(* PLC project CALENDARS, Actility iec61131 1.0.24, author Laurent Nicq *)
(* stored: creationDateTime 2013-03-20T17:09:43, version 1.0.1, modificationDateTime 2013-07-25T17:16:31 *)

PROGRAM Calendar_Single
  VAR
    Light_Outside : BOOL;
  END_VAR
  VAR_EXTERNAL
    TimeSTART_Single : TOD;
    TimeEND_Single : TOD;
    Date_Single : DATE;
  END_VAR
  VAR
    Calendar_Name : STRING := 'Evening';
  END_VAR

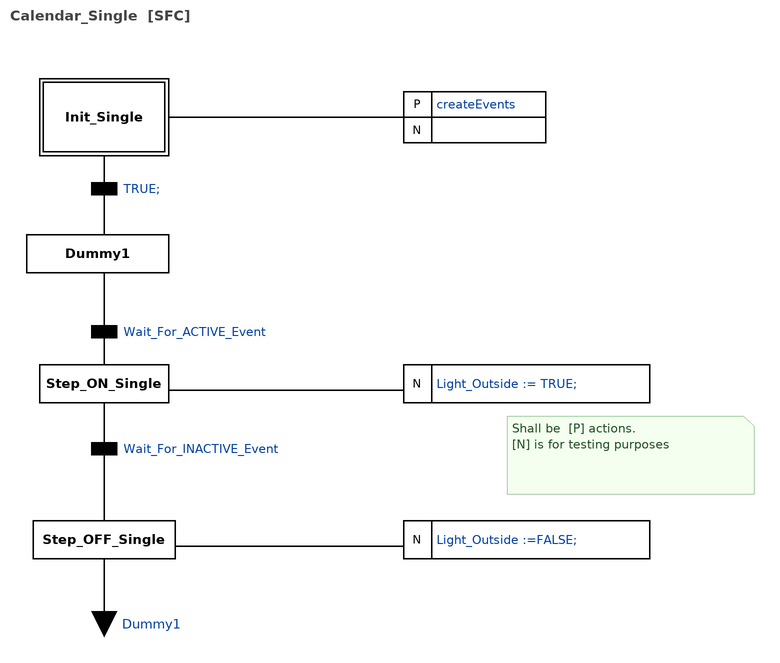
(* Shall be  [P] actions.
[N] is for testing purposes *)
INITIAL_STEP Init_Single:
  createEvents(P);
  (N);
END_STEP
TRANSITION FROM Init_Single TO Dummy1
  := TRUE;
END_TRANSITION
STEP Dummy1:
END_STEP
TRANSITION FROM Dummy1 TO Step_ON_Single  (* Wait_For_ACTIVE_Event *)
  := checkCalendarEvent (Calendar_Name);
END_TRANSITION
STEP Step_ON_Single:
  STEP_ON_SINGLE_INLINE1(N);
END_STEP
ACTION STEP_ON_SINGLE_INLINE1:
  Light_Outside := TRUE;
END_ACTION
TRANSITION FROM Step_ON_Single TO Step_OFF_Single  (* Wait_For_INACTIVE_Event *)
  := NOT(checkCalendarEvent (Calendar_Name) );
END_TRANSITION
STEP Step_OFF_Single:
  STEP_OFF_SINGLE_INLINE2(N);
END_STEP
ACTION STEP_OFF_SINGLE_INLINE2:
  Light_Outside :=FALSE;
END_ACTION

ACTION createEvents:
TimeEND_Single := ADD_TOD_TIME( TimeSTART_Single, T#1m0s);
newCalendarEvent (Calendar_Name, Date_Single, TimeSTART_Single, TimeEND_Single);
              
END_ACTION
END_PROGRAM

PROGRAM Calendar_Weekly
  VAR
    Light_Television : BOOL;
  END_VAR
  VAR_EXTERNAL
    TimeSTART_Single : TOD;
    TimeSTART_Weekly : TOD;
    TimeEND_Weekly : TOD;
  END_VAR
  VAR
    Calendar_Name : STRING := 'Movie';
  END_VAR
  VAR_EXTERNAL
    Days_Of_week : DINT;
  END_VAR

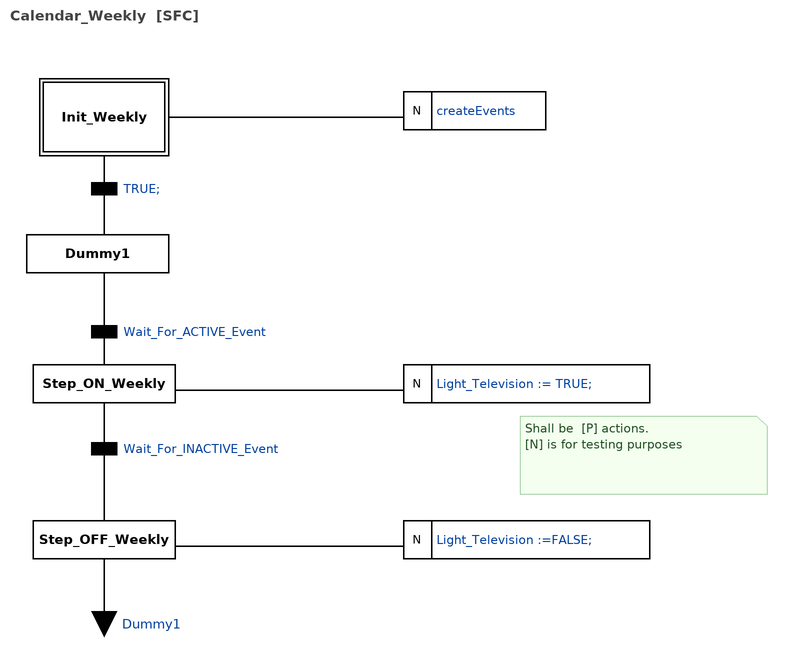
(* Shall be  [P] actions.
[N] is for testing purposes *)
INITIAL_STEP Init_Weekly:
  createEvents(N);
END_STEP
TRANSITION FROM Init_Weekly TO Dummy1
  := TRUE;
END_TRANSITION
STEP Dummy1:
END_STEP
TRANSITION FROM Dummy1 TO Step_ON_Weekly  (* Wait_For_ACTIVE_Event *)
  := checkCalendarEvent (Calendar_Name);
END_TRANSITION
STEP Step_ON_Weekly:
  STEP_ON_WEEKLY_INLINE1(N);
END_STEP
ACTION STEP_ON_WEEKLY_INLINE1:
  Light_Television := TRUE;
END_ACTION
TRANSITION FROM Step_ON_Weekly TO Step_OFF_Weekly  (* Wait_For_INACTIVE_Event *)
  := NOT(checkCalendarEvent (Calendar_Name) );
END_TRANSITION
STEP Step_OFF_Weekly:
  STEP_OFF_WEEKLY_INLINE2(N);
END_STEP
ACTION STEP_OFF_WEEKLY_INLINE2:
  Light_Television :=FALSE;
END_ACTION

ACTION createEvents:
TimeSTART_Weekly := ADD_TOD_TIME( TimeSTART_Single, T#4m0s);
TimeEND_Weekly := ADD_TOD_TIME( TimeSTART_Single, T#5m0s);
newCalendarWeeklyEvent (Calendar_Name, TimeSTART_Weekly, TimeEND_Weekly, Days_Of_week );
              
END_ACTION
END_PROGRAM

PROGRAM Calendar_Daily
  VAR
    Light_Kitchen : BOOL;
  END_VAR
  VAR_EXTERNAL
    TimeSTART_Daily : TOD;
    TimeSTART_Single : TOD;
    TimeEND_Daily : TOD;
  END_VAR
  VAR
    Calendar_Name : STRING := 'Dining';
  END_VAR
  VAR_EXTERNAL
    Days_Interval : DINT;
  END_VAR

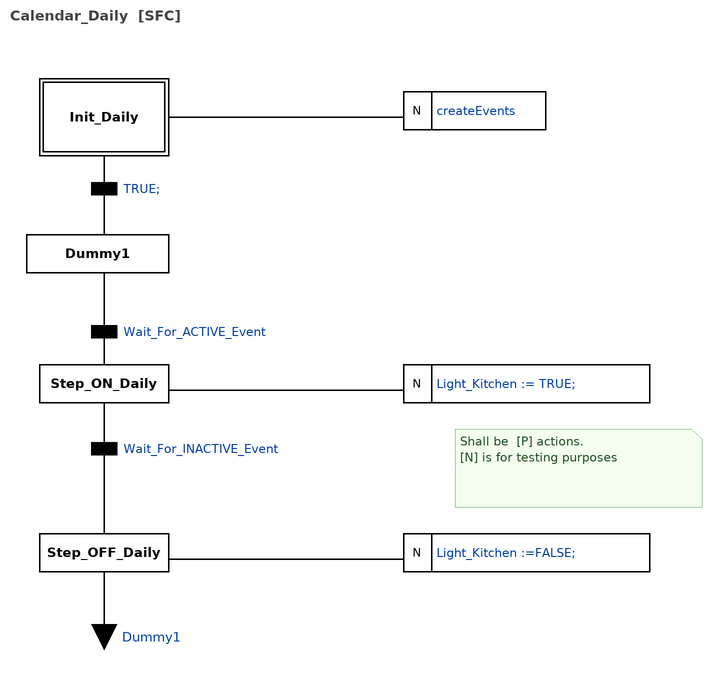
(* Shall be  [P] actions.
[N] is for testing purposes *)
INITIAL_STEP Init_Daily:
  createEvents(N);
END_STEP
TRANSITION FROM Init_Daily TO Dummy1
  := TRUE;
END_TRANSITION
STEP Dummy1:
END_STEP
TRANSITION FROM Dummy1 TO Step_ON_Daily  (* Wait_For_ACTIVE_Event *)
  := checkCalendarEvent (Calendar_Name);
END_TRANSITION
STEP Step_ON_Daily:
  STEP_ON_DAILY_INLINE1(N);
END_STEP
ACTION STEP_ON_DAILY_INLINE1:
  Light_Kitchen := TRUE;
END_ACTION
TRANSITION FROM Step_ON_Daily TO Step_OFF_Daily  (* Wait_For_INACTIVE_Event *)
  := NOT(checkCalendarEvent (Calendar_Name) );
END_TRANSITION
STEP Step_OFF_Daily:
  STEP_OFF_DAILY_INLINE2(N);
END_STEP
ACTION STEP_OFF_DAILY_INLINE2:
  Light_Kitchen :=FALSE;
END_ACTION

ACTION createEvents:
TimeSTART_Daily := ADD_TOD_TIME( TimeSTART_Single, T#2m0s);
TimeEND_Daily := ADD_TOD_TIME( TimeSTART_Single, T#3m0s);
newCalendarDailyEvent (Calendar_Name, TimeSTART_Daily, TimeEND_Daily, Days_Interval );
              
END_ACTION
END_PROGRAM

CONFIGURATION Astro_test
  RESOURCE main_config ON PLC
    VAR_GLOBAL
      Date_Single : DATE := DATE#2013-07-25;  (* adjust date for testing *)
      TimeSTART_Single : TOD := TOD#16:56:00;  (* adjust time for testing *)
      TimeEND_Single : TOD;  (* calculated for testing *)
      TimeSTART_Daily : TOD;  (* calculated for testing *)
      TimeEND_Daily : TOD;  (* calculated for testing *)
      Days_Interval : DINT := 1;  (* Every day (Daily Event) *)
      TimeSTART_Weekly : TOD;  (* calculated for testing *)
      TimeEND_Weekly : TOD;  (* calculated for testing *)
      Days_Of_week : DINT := 2#0111_1111;  (* All days (Weekly Event) *)
    END_VAR
    TASK task_main(INTERVAL := T#1s0ms, PRIORITY := 0);
    PROGRAM calendar1 WITH task_main : Calendar_Single;
    PROGRAM calendar2 WITH task_main : Calendar_Daily;
    PROGRAM calendar3 WITH task_main : Calendar_Weekly;
  END_RESOURCE
END_CONFIGURATION
